(* PLC project , CODESYS CODESYS V3.5 SP16 Patch 4 *)
(* stored: creationDateTime 2021-04-29T08:49:20.3586754, modificationDateTime 2021-04-29T00:03:20.8398477 *)

FUNCTION_BLOCK sf_equ_BaseTest_RandomTest_Res1 EXTENDS FB_TestSuite

            TC1();
          

METHOD TC1
  VAR_INPUT
    t_Active : BOOL := 1;
    t_ChannelA : BOOL := 0;
    t_ChannelB : BOOL := 1;
    t_DiscrepancyTime : TIME := TIME#37s785ms;
  END_VAR
  VAR
    Fun : sf_equ;
    Result1 : BOOL;
    Result2 : BOOL;
    Result3 : BOOL;
    ExpectedResult1 : BOOL := FALSE;
    ExpectedResult2 : BOOL := FALSE;
    ExpectedResult3 : BOOL := FALSE;
    Condition : BOOL;
  END_VAR
                  TEST('TC1');

Fun(Active := t_Active, ChannelA := t_ChannelA, ChannelB := t_ChannelB, DiscrepancyTime := t_DiscrepancyTime, Ready => Result1, EquivalentOut => Result2, Error => Result3);

AssertTrue(Condition := (Result1 = ExpectedResult1),
			Message := 'Result1 is True');
			
TEST_FINISHED();
                
END_METHOD
END_FUNCTION_BLOCK
